  rq_activate_all_grippers(False)
  # end: URCap Program Node
  $ 4 "MoveJ"
  $ 5 "Waypoint_1" "breakAfter"
  movej(pose_add(get_target_tcp_pose(), pose_sub(Waypoint_1_to_p, Waypoint_1_from_p)), a=1.3962634015954636, v=1.0471975511965976)
  $ 6 "Home"
  movej([-1.7469009394078796, -1.3843886428855203, -2.1469917153867106, -1.1815006968848882, 1.5786694858919006, 0.3920050440532714], a=1.3962634015954636, v=1.0471975511965976)
  $ 75 "Thread_1"
  thread Thread_1():
    while (True):
      $ 76 "Robot_Force≔force()"
      global Robot_Force= force ()
      $ 77 "If LL_Inintial≟ True "
      if (get_standard_digital_in(0) ==   True  ):
        $ 78 "Set LL_Light=On"
        set_standard_digital_out(0, True)
      else:
        $ 79 "Else" "noBreak"
        $ 80 "Set LL_Light=Off"
        set_standard_digital_out(0, False)
      end
      $ 81 "sync()"
      sync()
    end
  end
  threadId_Thread_1 = run Thread_1()
  $ 82 "Thread_2"
  thread Thread_2():
    while (True):
      $ 83 "If LR_Freedrive≟ True "
      if (get_standard_digital_in(1) ==   True  ):
        $ 84 "Set LR_Light=On"
        set_standard_digital_out(1, True)
      else:
        $ 85 "Else" "noBreak"
        $ 86 "Set LR_Light=Off"
        set_standard_digital_out(1, False)
      end
      $ 87 "sync()"
      sync()
    end
  end
  threadId_Thread_2 = run Thread_2()
  while (True):
    $ 7 "Robot Program"
    $ 8 "MoveJ"
    $ 9 "cycle_time: Reset"
    cycle_time = 0
    $ 10 "cycle_time: Start"
    cycle_time_is_counting = True
    # begin: URCap Program Node
    #   Source: Robotiq_Grippers, 1.8.7.10599, Robotiq Inc.
    #   Type: Gripper
    $ 11 "Gripper Move37mm (1)"
    if not(gripper_connected[0]):
      popup("Gripper 1 must be connected to run this program.", "No connection", False, True, True)
    end
    if not(rq_is_gripper_activated("1")):
      popup("Gripper 1 is not activated. Go to Installation tab > Gripper to activate it and run the program again.", "Not activated", False, True, True)
    end
    rq_set_pos_spd_for(67, 255, 0, "1")
    rq_wait_pos_spe_for_request(67, 255, 0, "1")
    rq_go_to("1")
    rq_wait("1")
    # end: URCap Program Node
    $ 12 "Unload"
    def Unload_trans(pose):
    return p[pose[0], pose[1], pose[2], 0, 0, 0]
  end
  def Unload_rot(pose):
  return p[0, 0, 0, pose[3], pose[4], pose[5]]
  end
  def Unload_compute_pallet_waypoint(T_base_feature_taught, T_feature_referencePoint_taught, T_referencePoint_approach_taught, T_base_feature, T_base_referencePoint):
  local trans_referencePoint_approach_in_feature_taught = pose_sub(Unload_trans(pose_trans(T_feature_referencePoint_taught, T_referencePoint_approach_taught)), Unload_trans(T_feature_referencePoint_taught))
  local rot_referencePoint_approach_in_feature_taught = pose_trans(Unload_rot(T_feature_referencePoint_taught), pose_trans(Unload_rot(T_referencePoint_approach_taught), pose_inv(Unload_rot(T_feature_referencePoint_taught))))
  T_feature_referencePoint = pose_trans(pose_inv(T_base_feature), T_base_referencePoint)
  rot_referencePoint_approach = pose_trans(pose_inv(Unload_rot(T_feature_referencePoint)), pose_trans(rot_referencePoint_approach_in_feature_taught, Unload_rot(T_feature_referencePoint)))
  T_feature_approach = pose_trans(trans_referencePoint_approach_in_feature_taught, pose_trans(T_feature_referencePoint, rot_referencePoint_approach))
  T_base_approach = pose_trans(T_base_feature, T_feature_approach)
  return T_base_approach
  end
  Pallet_1_tct = 6
  if (Pallet_1_cnt > 6 or Pallet_1_cnt < 1):
    Pallet_1_cnt = 1
  end
  $ 13 "Patterns" "noBreak"
  $ 14 "Grid_Pattern_1" "noBreak"
  $ 19 "Layers" "noBreak"
  if (Pallet_1_cnt < 7):
    Pallet_1_lno = 1
    Pallet_1_lct = Pallet_1_cnt
    global CornerItem_1=pose_trans(p[0.0,0.0,0.0,0.0,0.0,0.0], pose_trans(p[-.000000000000, -.000000000000, -.000000000000, .000000000000, .000000000000, .000000000000], p[.316711535192, -.318531249341, -.031450600752, .607306623548, 3.082311525429, -.000520031619]))
    global CornerItem_2=pose_trans(p[0.0,0.0,0.0,0.0,0.0,0.0], pose_trans(p[-.000000000000, -.000000000000, -.000000000000, .000000000000, .000000000000, .000000000000], p[.316447335533, -.379133905457, -.030769187293, .607278067865, 3.082046644026, -.000655612285]))
    global CornerItem_3=pose_trans(p[0.0,0.0,0.0,0.0,0.0,0.0], pose_trans(p[-.000000000000, -.000000000000, -.000000000000, .000000000000, .000000000000, .000000000000], p[.437520916762, -.379468851622, -.029561984544, .607124757147, 3.081932793043, -.000677010974]))
    global CornerItem_4=pose_trans(p[0.0,0.0,0.0,0.0,0.0,0.0], pose_trans(p[-.000000000000, -.000000000000, -.000000000000, .000000000000, .000000000000, .000000000000], p[.435990378353, -.317372949526, -.031448303994, .607223711556, 3.082018242770, -.000628895936]))
    Pallet_1_cnt_x = (Pallet_1_lct - 1) % 2
    Pallet_1_cnt_y = floor((Pallet_1_lct - 1) / 2)
    referencePoint = interpolate_pose(interpolate_pose(CornerItem_1, CornerItem_2, Pallet_1_cnt_x/1), interpolate_pose(CornerItem_4, CornerItem_3,Pallet_1_cnt_x/1), Pallet_1_cnt_y/2)
    direction = p[0,0,1,0,0,0]
    referencePoint = pose_add (referencePoint,p[0.0*direction[0],0.0*direction[1],0.0*direction[2],0,0,0])
  end
  Approach_p = Unload_compute_pallet_waypoint(p[0.0,0.0,0.0,0.0,0.0,0.0], pose_trans(pose_inv(p[0.0,0.0,0.0,0.0,0.0,0.0]), p[0.31671153519228795,-0.31853124934123117,-0.031450600751847135,0.6073066235480151,3.0823115254293114,-5.200316192790575E-4]), p[1.3092328866926017E-5,-5.506968575502702E-5,-0.09343729629070505,-1.1467826098044958E-5,2.8421636282015192E-5,4.183498516292272E-5], p[0.0,0.0,0.0,0.0,0.0,0.0], referencePoint)
  Approach_p = pose_trans(p[0.31671153519228795,-0.31853124934123117,-0.031450600751847135,0.6073066235480162,3.0823115254293114,-5.200316201336444E-4], pose_trans(pose_inv(referencePoint), Approach_p))
  ToolActionPoint_p = Unload_compute_pallet_waypoint(p[0.0,0.0,0.0,0.0,0.0,0.0], pose_trans(pose_inv(p[0.0,0.0,0.0,0.0,0.0,0.0]), p[0.31671153519228795,-0.31853124934123117,-0.031450600751847135,0.6073066235480151,3.0823115254293114,-5.200316192790575E-4]), p[0.0,0.0,0.0,0.0,0.0,0.0], p[0.0,0.0,0.0,0.0,0.0,0.0], referencePoint)
  ToolActionPoint_p = pose_trans(p[0.31671153519228795,-0.31853124934123117,-0.031450600751847135,0.6073066235480162,3.0823115254293114,-5.200316201336444E-4], pose_trans(pose_inv(referencePoint), ToolActionPoint_p))
  Exit_1_p = Unload_compute_pallet_waypoint(p[0.0,0.0,0.0,0.0,0.0,0.0], pose_trans(pose_inv(p[0.0,0.0,0.0,0.0,0.0,0.0]), p[0.31671153519228795,-0.31853124934123117,-0.031450600751847135,0.6073066235480151,3.0823115254293114,-5.200316192790575E-4]), p[-1.5117529851171874E-5,-4.952688991535781E-5,-0.09342286897399588,-3.0088363799123978E-5,-3.1453721294772E-5,8.58589236342157E-5], p[0.0,0.0,0.0,0.0,0.0,0.0], referencePoint)
  Exit_1_p = pose_trans(p[0.31671153519228795,-0.31853124934123117,-0.031450600751847135,0.6073066235480162,3.0823115254293114,-5.200316201336444E-4], pose_trans(pose_inv(referencePoint), Exit_1_p))
  $ 20 "At Each Item" "noBreak"
  $ 21 "Generated Movements" "noBreak"
  $ 22 "MoveJ" "noBreak"
  $ 23 "Approach" "noBreak"
  movej(get_inverse_kin(pose_trans(referencePoint, pose_trans(p[.413867348153, .174574952464, -.031541999354, -.607306623547, -3.082311525424, .000520031624], Approach_p)), qnear=Approach_q), a=1.3962634015954636, v=1.0471975511965976, r=0.01)
  $ 24 "MoveL" "noBreak"
  $ 25 "ToolActionPoint" "noBreak"
  movel(pose_trans(referencePoint, pose_trans(p[.413867348153, .174574952464, -.031541999354, -.607306623547, -3.082311525424, .000520031624], ToolActionPoint_p)), a=1.2, v=0.25)
  $ 26 "Tool action" "noBreak"
  # begin: URCap Program Node
  #   Source: Robotiq_Grippers, 1.8.7.10599, Robotiq Inc.
  #   Type: Gripper
  $ 27 "Gripper Close (1)" "noBreak"
  if not(gripper_connected[0]):
    popup("Gripper 1 must be connected to run this program.", "No connection", False, True, True)
  end
  if not(rq_is_gripper_activated("1")):
    popup("Gripper 1 is not activated. Go to Installation tab > Gripper to activate it and run the program again.", "Not activated", False, True, True)
  end
  rq_set_pos_spd_for(255, 255, 77, "1")
  rq_wait_pos_spe_for_request(255, 255, 77, "1")
  rq_go_to("1")
  rq_wait("1")
  # end: URCap Program Node
  $ 28 "MoveL" "noBreak"
  $ 29 "Exit_1" "noBreak"
  movel(pose_trans(referencePoint, pose_trans(p[.413867348153, .174574952464, -.031541999354, -.607306623547, -3.082311525424, .000520031624], Exit_1_p)), a=1.2, v=0.25, r=0.015)
  Pallet_1_sep = False
  if (Pallet_1_cnt >= 6):
    Pallet_1_cnt = 1
  else:
    Pallet_1_cnt = Pallet_1_cnt + 1
  end
  $ 30 "Conveyor_Trans" "breakAfter"
  movej(get_inverse_kin(Conveyor_Trans_p, qnear=Conveyor_Trans_q), a=1.3962634015954636, v=1.0471975511965976, r=0.05)
  $ 31 "Conv_Drop_Entry" "breakAfter"
  movej(get_inverse_kin(Conv_Drop_Entry_p, qnear=Conv_Drop_Entry_q), a=1.3962634015954636, v=1.0471975511965976, r=0.043)
  $ 32 "Conveyor_Drop" "breakAfter"
  movej(get_inverse_kin(Conveyor_Drop_p, qnear=Conveyor_Drop_q), a=1.3962634015954636, v=1.0471975511965976)
  $ 33 "Set Payload: Hande_Payload"
  set_target_payload(1.320000, [-0.001000, -0.005000, 0.062000], [0.002445, 0.002445, 0.002445, 0.000000, 0.000000, 0.000000])
  # begin: URCap Program Node
  #   Source: Robotiq_Grippers, 1.8.7.10599, Robotiq Inc.
  #   Type: Gripper
  $ 34 "Gripper Move37mm (1)"
  if not(gripper_connected[0]):
    popup("Gripper 1 must be connected to run this program.", "No connection", False, True, True)
  end
  if not(rq_is_gripper_activated("1")):
    popup("Gripper 1 is not activated. Go to Installation tab > Gripper to activate it and run the program again.", "Not activated", False, True, True)
  end
  rq_set_pos_spd_for(67, 255, 77, "1")
  rq_wait_pos_spe_for_request(67, 255, 77, "1")
  rq_go_to("1")
  rq_wait("1")
  # end: URCap Program Node
  $ 35 "Conv_Drop_Entry" "breakAfter"
  movej(get_inverse_kin(Conv_Drop_Entry_p, qnear=Conv_Drop_Entry_q), a=1.3962634015954636, v=1.0471975511965976, r=0.01)
  $ 36 "Wait Left_Sensor=HI"
  while (get_standard_digital_in(5) == False):
    sync()
  end
  $ 37 "Set Run_Conveyor=On"
  set_standard_digital_out(3, True)
  $ 38 "Conv_Pick_Entry" "breakAfter"
  movej(get_inverse_kin(Conv_Pick_Entry_p, qnear=Conv_Pick_Entry_q), t=4.0, r=0.015)
  $ 39 "Conv_Pick" "breakAfter"
  movej(get_inverse_kin(Conv_Pick_p, qnear=Conv_Pick_q), a=1.3962634015954636, v=1.0471975511965976)
  $ 40 "Wait Right_Sensor=HI"
  while (get_standard_digital_in(4) == False):
    sync()
  end
  $ 41 "Wait: 0.3"
  sleep(0.3)
  $ 42 "Set Run_Conveyor=Off"
  set_standard_digital_out(3, False)
  # begin: URCap Program Node
  #   Source: Robotiq_Grippers, 1.8.7.10599, Robotiq Inc.
  #   Type: Gripper
  $ 43 "Gripper Close (1)"
  if not(gripper_connected[0]):
    popup("Gripper 1 must be connected to run this program.", "No connection", False, True, True)
  end
  if not(rq_is_gripper_activated("1")):
    popup("Gripper 1 is not activated. Go to Installation tab > Gripper to activate it and run the program again.", "Not activated", False, True, True)
  end
  rq_set_pos_spd_for(255, 255, 77, "1")
  rq_wait_pos_spe_for_request(255, 255, 77, "1")
  rq_go_to("1")
  rq_wait("1")
  # end: URCap Program Node
  $ 44 "Conv_Pick_Entry" "breakAfter"
  movej(get_inverse_kin(Conv_Pick_Entry_p, qnear=Conv_Pick_Entry_q), a=1.3962634015954636, v=1.0471975511965976, r=0.01)
  $ 45 "If Cycle_Count≟3"
  if (Cycle_Count == 3):
    $ 46 "Call SubProgram_1"
    SubProgram_1()
  end
  $ 47 "Pallet_Load"
  def Pallet_Load_trans(pose):
  return p[pose[0], pose[1], pose[2], 0, 0, 0]
  end
  def Pallet_Load_rot(pose):
  return p[0, 0, 0, pose[3], pose[4], pose[5]]
  end
  def Pallet_Load_compute_pallet_waypoint(T_base_feature_taught, T_feature_referencePoint_taught, T_referencePoint_approach_taught, T_base_feature, T_base_referencePoint):
  local trans_referencePoint_approach_in_feature_taught = pose_sub(Pallet_Load_trans(pose_trans(T_feature_referencePoint_taught, T_referencePoint_approach_taught)), Pallet_Load_trans(T_feature_referencePoint_taught))
  local rot_referencePoint_approach_in_feature_taught = pose_trans(Pallet_Load_rot(T_feature_referencePoint_taught), pose_trans(Pallet_Load_rot(T_referencePoint_approach_taught), pose_inv(Pallet_Load_rot(T_feature_referencePoint_taught))))
  T_feature_referencePoint = pose_trans(pose_inv(T_base_feature), T_base_referencePoint)
  rot_referencePoint_approach = pose_trans(pose_inv(Pallet_Load_rot(T_feature_referencePoint)), pose_trans(rot_referencePoint_approach_in_feature_taught, Pallet_Load_rot(T_feature_referencePoint)))
  T_feature_approach = pose_trans(trans_referencePoint_approach_in_feature_taught, pose_trans(T_feature_referencePoint, rot_referencePoint_approach))
  T_base_approach = pose_trans(T_base_feature, T_feature_approach)
  return T_base_approach
  end
  Pallet_1_tct_1 = 6
  if (Pallet_1_cnt_1 > 6 or Pallet_1_cnt_1 < 1):
    Pallet_1_cnt_1 = 1
  end
  $ 48 "Patterns" "noBreak"
  $ 49 "Grid_Pattern_2" "noBreak"
  $ 54 "Layers" "noBreak"
  if (Pallet_1_cnt_1 < 7):
    Pallet_1_lno_1 = 1
    Pallet_1_lct_1 = Pallet_1_cnt_1
    global CornerItem_5=pose_trans(p[0.0,0.0,0.0,0.0,0.0,0.0], pose_trans(p[-.000000000000, -.000000000000, -.000000000000, .000000000000, .000000000000, .000000000000], p[.316724873388, -.318532854525, -.031439387103, .607248458166, 3.082309862675, -.000526581507]))
    global CornerItem_6=pose_trans(p[0.0,0.0,0.0,0.0,0.0,0.0], pose_trans(p[-.000000000000, -.000000000000, -.000000000000, .000000000000, .000000000000, .000000000000], p[.316502308265, -.381006139800, -.030709140063, .607126482619, 3.081951252629, -.000716299029]))
    global CornerItem_7=pose_trans(p[0.0,0.0,0.0,0.0,0.0,0.0], pose_trans(p[-.000000000000, -.000000000000, -.000000000000, .000000000000, .000000000000, .000000000000], p[.437535841516, -.380982637874, -.029533361096, .606971215985, 3.081950779676, -.000656559810]))
    global CornerItem_8=pose_trans(p[0.0,0.0,0.0,0.0,0.0,0.0], pose_trans(p[-.000000000000, -.000000000000, -.000000000000, .000000000000, .000000000000, .000000000000], p[.435972496869, -.317364952014, -.031463786887, .607213200201, 3.082067925394, -.000614784866]))
    Pallet_1_cnt_1_x = (Pallet_1_lct_1 - 1) % 2
    Pallet_1_cnt_1_y = floor((Pallet_1_lct_1 - 1) / 2)
    referencePoin_1 = interpolate_pose(interpolate_pose(CornerItem_5, CornerItem_6, Pallet_1_cnt_1_x/1), interpolate_pose(CornerItem_8, CornerItem_7,Pallet_1_cnt_1_x/1), Pallet_1_cnt_1_y/2)
    direction = p[0,0,1,0,0,0]
    referencePoin_1 = pose_add (referencePoin_1,p[0.0*direction[0],0.0*direction[1],0.0*direction[2],0,0,0])
  end
  Approach_1_p = Pallet_Load_compute_pallet_waypoint(p[0.0,0.0,0.0,0.0,0.0,0.0], pose_trans(pose_inv(p[0.0,0.0,0.0,0.0,0.0,0.0]), p[0.3167248733883772,-0.31853285452466895,-0.031439387102959626,0.6072484581664501,3.082309862674719,-5.265815066939557E-4]), p[-2.618897918105212E-5,-3.512210748626843E-5,-0.09343291427718783,-2.9477256378669938E-5,-3.4581789295188886E-5,1.4630890742805435E-5], p[0.0,0.0,0.0,0.0,0.0,0.0], referencePoin_1)
  Approach_1_p = pose_trans(p[0.3167248733883772,-0.31853285452466895,-0.031439387102959626,0.6072484581664518,3.082309862674719,-5.265815051792499E-4], pose_trans(pose_inv(referencePoin_1), Approach_1_p))
  ToolActionPoi_1_p = Pallet_Load_compute_pallet_waypoint(p[0.0,0.0,0.0,0.0,0.0,0.0], pose_trans(pose_inv(p[0.0,0.0,0.0,0.0,0.0,0.0]), p[0.3167248733883772,-0.31853285452466895,-0.031439387102959626,0.6072484581664501,3.082309862674719,-5.265815066939557E-4]), p[-5.551115123125783E-17,-2.7755575615628914E-17,0.0,1.5601363517053764E-12,-3.0736403819255765E-13,-1.5820678597216844E-15], p[0.0,0.0,0.0,0.0,0.0,0.0], referencePoin_1)
  ToolActionPoi_1_p = pose_trans(p[0.3167248733883772,-0.31853285452466895,-0.031439387102959626,0.6072484581664518,3.082309862674719,-5.265815051792499E-4], pose_trans(pose_inv(referencePoin_1), ToolActionPoi_1_p))
  Exit_2_p = Pallet_Load_compute_pallet_waypoint(p[0.0,0.0,0.0,0.0,0.0,0.0], pose_trans(pose_inv(p[0.0,0.0,0.0,0.0,0.0,0.0]), p[0.3167248733883772,-0.31853285452466895,-0.031439387102959626,0.6072484581664501,3.082309862674719,-5.265815066939557E-4]), p[-3.090263950372707E-5,-3.20921088760584E-5,-0.09344157968440611,-9.274250718455154E-6,-6.1135349402295215E-6,-8.106809517786809E-6], p[0.0,0.0,0.0,0.0,0.0,0.0], referencePoin_1)
  Exit_2_p = pose_trans(p[0.3167248733883772,-0.31853285452466895,-0.031439387102959626,0.6072484581664518,3.082309862674719,-5.265815051792499E-4], pose_trans(pose_inv(referencePoin_1), Exit_2_p))
  $ 55 "At Each Item" "noBreak"
  $ 56 "Generated Movements" "noBreak"
  $ 57 "MoveJ" "noBreak"
  $ 58 "Approach_1" "noBreak"
  movej(get_inverse_kin(pose_trans(referencePoin_1, pose_trans(p[.413873568837, .174586282196, -.031536629224, -.607248458166, -3.082309862675, .000526581505], Approach_1_p)), qnear=Approach_1_q), a=1.3962634015954636, v=1.0471975511965976, r=0.015)
  $ 59 "MoveL" "noBreak"
  $ 60 "ToolActionPoi_1" "noBreak"
  movel(pose_trans(referencePoin_1, pose_trans(p[.413873568837, .174586282196, -.031536629224, -.607248458166, -3.082309862675, .000526581505], ToolActionPoi_1_p)), a=1.2, v=0.25)
  $ 61 "Tool action" "noBreak"
  # begin: URCap Program Node
  #   Source: Robotiq_Grippers, 1.8.7.10599, Robotiq Inc.
  #   Type: Gripper
  $ 62 "Gripper Move37mm (1)" "noBreak"
  if not(gripper_connected[0]):
    popup("Gripper 1 must be connected to run this program.", "No connection", False, True, True)
  end
  if not(rq_is_gripper_activated("1")):
    popup("Gripper 1 is not activated. Go to Installation tab > Gripper to activate it and run the program again.", "Not activated", False, True, True)
  end
  rq_set_pos_spd_for(67, 255, 77, "1")
  rq_wait_pos_spe_for_request(67, 255, 77, "1")
  rq_go_to("1")
  rq_wait("1")
  # end: URCap Program Node
  $ 63 "MoveL" "noBreak"
  $ 64 "Exit_2" "noBreak"
  movel(pose_trans(referencePoin_1, pose_trans(p[.413873568837, .174586282196, -.031536629224, -.607248458166, -3.082309862675, .000526581505], Exit_2_p)), a=1.2, v=0.25)
  $ 65 "Action after palletizing" "noBreak"
  if (Pallet_1_cnt_1 == 6):
    $ 66 "Home" "noBreak"
    movej([-1.7469009394078796, -1.3843886428855203, -2.1469917153867106, -1.1815006968848882, 1.5786694858919006, 0.3920050440532714], a=1.3962634015954636, v=1.0471975511965976)
    $ 67 "Halt" "noBreak"
    halt
  end
  Pallet_1_sep_1 = False
  if (Pallet_1_cnt_1 >= 6):
    Pallet_1_cnt_1 = 1
  else:
    Pallet_1_cnt_1 = Pallet_1_cnt_1 + 1
  end
  $ 68 "cycle_time: Stop"
  cycle_time_is_counting = False
  $ 69 "Cycle_Count≔Cycle_Count+1"
  global Cycle_Count=Cycle_Count+1
  end
end
